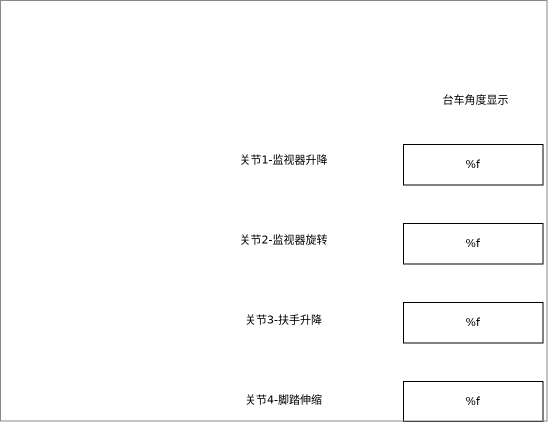
VISUALIZATION motRangeCar  // 548x422
    Label (403,86 145x28), "台车角度显示"
    Label (211,146 145x28), "关节1-监视器升降"
    Label (211,226 145x28), "关节2-监视器旋转"
    Label (211,306 145x28), "关节3-扶手升降"
    Label (211,386 145x28), "关节4-脚踏伸缩"
    Rectangle (403,144 140x41), "%f", text variable: g_systemInfo.m_cartInfo.m_curJntPosDegMM[1]
    Rectangle (403,223 140x41), "%f", text variable: g_systemInfo.m_cartInfo.m_curJntPosDegMM[2]
    Rectangle (403,302 140x41), "%f", text variable: g_systemInfo.m_cartInfo.m_curJntPosDegMM[3]
    Rectangle (403,381 140x41), "%f", text variable: g_systemInfo.m_cartInfo.m_curJntPosDegMM[4]
END_VISUALIZATION

(* stored: Version 1.1.0.1, ProductVersion 3.1.4024.11
   Visu motRangeCar: Id {b7fecb6d-4394-49ac-8e05-b25fab64cd46} *)
